KUKA KRL program: chk_w6_wechs_ok.src

&ACCESS RV3
&COMMENT Gripper Accelo Teto
DEF chk_w6_wechs_ok( )

; VERIFICAÇÃO DE FERRAMENTA: Gripper Teto Accelo

$TIMER[10] = 0
$TIMER_STOP[10] = FALSE

wait for (($IN[585]) and ($IN[577]) and ($in[161]) and ($in[177])and ($in[193]) and ($in[201]) and ($in[209]) and ($IN[169]) and (not $in[185]) AND ($in[219]))

$TIMER_STOP[10] = TRUE
$TIMER[10] = 0

;//---- End -------
;Diag_Appl(#Off,5)

END
